FUNCTION F_DH : BOOL
VAR_INPUT
	theta : LREAL;
	d : LREAL;
	a : LREAL;
	alpha : LREAL;
	F_DH_OUT : REFERENCE TO FB_Matrix4x4;
END_VAR
VAR
END_VAR


F_DH_OUT.SetRC(0, 0, COS(theta));
F_DH_OUT.SetRC(0, 1, -SIN(theta)*COS(alpha));
F_DH_OUT.SetRC(0, 2, SIN(theta)*SIN(alpha));
F_DH_OUT.SetRC(0, 3, a*COS(theta));

F_DH_OUT.SetRC(1, 0, SIN(theta));
F_DH_OUT.SetRC(1, 1, COS(theta)*COS(alpha));
F_DH_OUT.SetRC(1, 2, -COS(theta)*SIN(alpha));
F_DH_OUT.SetRC(1, 3, a*SIN(theta));


F_DH_OUT.SetRC(2, 0, 0);
F_DH_OUT.SetRC(2, 1, SIN(alpha));
F_DH_OUT.SetRC(2, 2, COS(alpha));
F_DH_OUT.SetRC(2, 3, d);

F_DH_OUT.SetRC(3, 0, 0);
F_DH_OUT.SetRC(3, 1, 0);
F_DH_OUT.SetRC(3, 2, 0);
F_DH_OUT.SetRC(3, 3, 1);

END_FUNCTION

(* stored: Version 1.1.0.1, ProductVersion 3.1.4024.9
   POU F_DH: Id {dee419d7-6482-4789-b74f-e082a72f92a1}, SpecialFunc None *)
